Staubli VAL3: trigger.pgx

public program trigger(num x_nCamID (dimensions=1), bool& x_bError[] (dimensions=1))
begin
  //-----------------------------------------------------------------------
  //Header begin
  //Description of program
  // Acquire a new image and evaluate it on the camera.
  //
  //Input parameters
  //  num x_nCamID :
  //    role : camera's ID
  //
  //Output parameters
  //  bool x_bError :
  //    role : returns true if an error occurred and false otherwise
  //
  //Examples
  //  call trigger(nCamID,l_bError)
  //
  //History
  //  Creation : 19-05-08 - f.Rob
  //Header end
  //-----------------------------------------------------------------------

  //Trigger image acquire and evaluation
  call setEventAndWait(x_nCamID,8,x_bError)
end
